// TIA Portal V16 export
// export: Created 2022-01-26T18:31:05.3448932Z, ExportSetting WithDefaults, DisplayName Totally Integrated Automation Portal, DisplayVersion V16, DisplayName TIA Portal Version Control Interface, DisplayVersion V16, DisplayName TIA Portal Openness, DisplayVersion V16, DisplayName STEP 7 Professional, DisplayVersion V16, DisplayName STEP 7 Safety, DisplayVersion V16, DisplayName WinCC Advanced, DisplayVersion V16
VAR_GLOBAL   // PLC tag table "Default tag table"
   Tag_1 AT %M10.0 : Bool;
   Tag_2 AT %M10.1 : Bool;
   Tag_3 AT %M10.5 : Bool;
   Tag_4 AT %M10.6 : Bool;
   Tag_5 AT %M10.7 : Bool;
   Tag_6 AT %M11.0 : Bool;
END_VAR
